FUNCTION_BLOCK FB_RAMP
VAR_INPUT
	realRampInput: REAL;		(* input value *)
	mEnableRamp: BOOL;			(* bit=0:Output=Input, bit=1: Ramp active, mZeroOutout has higher priority *)
	mZeroOutput:BOOL;			(* bit=0 normal operation, bit=1 output zero *)
	realRampSpeed: REAL;		(* speed value/second *)
	realRampSampleTime: REAL; 	(* based on 100ns increments *)
	realEqualize: REAL;
END_VAR
VAR_OUTPUT
	realRampOutput: REAL;		(* output value *)
	mRampSaturised: BOOL;		(* ramp on the end *)
END_VAR

VAR
END_VAR

IF mEnableRamp AND NOT mZeroOutput THEN
	IF ABS(realRampOutput-realRampInput)<realEqualize THEN
		realRampOutput:=realRampInput; (* direct *)
		mRampSaturised:=TRUE;
	ELSE
		IF realRampOutput<realRampInput THEN (* increment *)
			realRampOutput:=realRampOutput+realRampSpeed*realRampSampleTime; (* realSampleTime in s *)
		END_IF
		IF realRampOutput>realRampInput THEN (* decrement *)
			realRampOutput:=realRampOutput-realRampSpeed*realRampSampleTime; (* realSampleTime in s *)
		END_IF
		mRampSaturised:=FALSE;
	END_IF
ELSE
	IF mZeroOutput THEN
		realRampOutput:=0;
	ELSE
		realRampOutput:=realRampInput; (* direct *)
	END_IF
END_IF

END_FUNCTION_BLOCK

(* stored: Version 1.1.0.1, ProductVersion 3.1.4024.11
   POU FB_RAMP: Id {5e240f73-e6b9-42ba-94ed-d31e5a6c6167}, SpecialFunc None *)
